TYPE st_AutoMode_AllocatingJob_1 :
STRUCT
	PickingNeedleInfo			: Array[0..3] OF st_AllocatingNeedleInfo;	//取針資料
	PlacingNeedleInfo			: ARRAY[0..3] OF st_AllocatingNeedleInfo;	//放針資料
	FastMode					: BOOL;
	SyncMode					: BOOL;
	HandShake					: st_HandshakeBase;
END_STRUCT
END_TYPE

(* stored: Version 1.1.0.1, ProductVersion 3.1.4024.13
   DUT st_AutoMode_AllocatingJob_1: Id {10ba63ae-b756-43bf-ad22-02b0e6c53c1e} *)
